// TIA Portal V21 export
VAR_GLOBAL   // PLC tag table "Comuni"
END_VAR
VAR_GLOBAL CONSTANT   // user constants
   StatoCmd_Stop : Byte := 0;
   StatoCmd_Auto : Byte := 1;
   StatoCmd_ManPos : Byte := 2;
   StatoCmd_ManNeg : Byte := 3;
   "StatoCmd_Scarico/Folle" : Byte := 4;
END_VAR
